{attribute 'pack_mode' := '1'} 
// ------------------------------------------------------------------------- 
//  SRCI Robot Library                                                
// ------------------------------------------------------------------------- 
//                                                                           
//  Object:      vAxesGroupCyclicOptionalDataPlcToRob                                       
//  Author:      Thorsten Brach                                                
//  Date:        2024-06-01
//
//  Description:                                              
//   
//                                                                           
//  Copyright: 
//    (C) 2024 Thorsten Brach. All rights reserved                                                                         
//                                                                           
//  Disclaimer:                                                                           
//    This project is provided without any guarantee and can be used for   
//    private and commercial purposes. Any commercial use is at the user’s 
//    own risk and responsibility.
//
// -------------------------------------------------------------------------
TYPE AxesGroupCyclicOptionalDataPlcToRob :
STRUCT
  /// Transmit cyclic data from PLC to RC for the usage in a subprogram on the RC called via the function “CallSubprogram”
  SubProgramData        :  AxesGroupCyclicOptionalDataSubProgram;
  /// short cartesian position with TCP position (X, Y,Z), rotation (RX, RY, RZ), configuration bytes (Config, TurnNumber), position of first external axis (E1) and corresponding coordinate systems (ToolNo, FrameNo)
  CartesianPosition     :  AxesGroupCyclicOptionalDataCartesianPosition;
  /// the external axis values for an extended cartesian position (E2, E3, E4, E5, E6) 
  /// When selected, Tool and Frame will automatically cyclically be sent from client to server.
  CartesianPositionExt  :  AxesGroupCyclicOptionalDataCartesianPositionExt;
  /// short axes position with joint values (J1, J2, J3,J4, J5, J6) and position of first external axis (E1)
  JointPosition         :  AxesGroupCyclicOptionalDataJointPosition;
  /// the external axis values for an extended joint position (E2, E3, E4, E5, E6)
  JointPositionExt      :  AxesGroupCyclicOptionalDataJointPositionExt;
  /// force with the divided forces in the individual directions (X, Y, Z, RX, RY, RZ)
  CartesianForce        :  AxesGroupCyclicOptionalDataCartesianForce;
  /// current force for the external axis (E1, E2, E3, E4, E5, E6)
  CartesianForceExt     :  AxesGroupCyclicOptionalDataCartesianForceExt;
END_STRUCT
END_TYPE

{attribute 'pack_mode' := '1'} 
// ------------------------------------------------------------------------- 
//  SRCI Robot Library                                                
// ------------------------------------------------------------------------- 
//                                                                           
//  Object:      AxesGroupCyclicOptionalDataRobToPlc                                       
//  Author:      Thorsten Brach                                                
//  Date:        2024-06-01
//
//  Description:                                              
//   
//                                                                           
//  Copyright: 
//    (C) 2024 Thorsten Brach. All rights reserved                                                                         
//                                                                           
//  Disclaimer:                                                                           
//    This project is provided without any guarantee and can be used for   
//    private and commercial purposes. Any commercial use is at the user’s 
//    own risk and responsibility.
//
// -------------------------------------------------------------------------
TYPE AxesGroupCyclicOptionalDataRobToPlc :
STRUCT
  /// Transmit cyclic data from PLC to RC for the usage in a subprogram on the RC called via the function “CallSubprogram”
  SubProgramData        :  AxesGroupCyclicOptionalDataSubProgram;
  /// short cartesian position with TCP position (X, Y,Z), rotation (RX, RY, RZ), configuration bytes (Config, TurnNumber), position of first external axis (E1) and corresponding coordinate systems (ToolNo, FrameNo)
  CartesianPosition     :  AxesGroupCyclicOptionalDataCartesianPosition;
  /// the external axis values for an extended cartesian position (E2, E3, E4, E5, E6) 
  /// When selected, Tool and Frame will automatically cyclically be sent from client to server.
  CartesianPositionExt  :  AxesGroupCyclicOptionalDataCartesianPositionExt;
  /// short axes position with joint values (J1, J2, J3,J4, J5, J6) and position of first external axis (E1)
  JointPosition         :  AxesGroupCyclicOptionalDataJointPosition;
  /// the external axis values for an extended joint position (E2, E3, E4, E5, E6)
  JointPositionExt      :  AxesGroupCyclicOptionalDataJointPositionExt;
  /// force with the divided forces in the individual directions (X, Y, Z, RX, RY, RZ)
  CartesianForce        :  AxesGroupCyclicOptionalDataCartesianForce;
  /// current force for the external axis (E1, E2, E3, E4, E5, E6)
  CartesianForceExt     :  AxesGroupCyclicOptionalDataCartesianForceExt;
  /// ctual axes current of individual axes (J1, J2, J3, J4, J5, J6)
  JointCurrent          :  AxesGroupCyclicOptionalDataJointCurrent;
  /// actual current for the external axis (E1, E2,E3, E4, E5, E6)
  JointCurrentExt       :  AxesGroupCyclicOptionalDataJointCurrentExt;  
END_STRUCT
END_TYPE

{attribute 'pack_mode' := '1'} 
// ------------------------------------------------------------------------- 
//  SRCI Robot Library                                                
// ------------------------------------------------------------------------- 
//                                                                           
//  Object:      AxesGroupCyclic                                       
//  Author:      Thorsten Brach                                                
//  Date:        2024-06-01
//
//  Description:                                              
//   
//                                                                           
//  Copyright: 
//    (C) 2024 Thorsten Brach. All rights reserved                                                                         
//                                                                           
//  Disclaimer:                                                                           
//    This project is provided without any guarantee and can be used for   
//    private and commercial purposes. Any commercial use is at the user’s 
//    own risk and responsibility.
//
// -------------------------------------------------------------------------
TYPE AxesGroupCyclic :
STRUCT
  /// Cyclic data from PLC to Robot 
  PlcToRob : AxesGroupCyclicPlcToRob;
  /// Cyclic data from Robot to PLC
  RobToPlc : AxesGroupCyclicRobToPlc;
END_STRUCT
END_TYPE

{attribute 'pack_mode' := '1'} 
// ------------------------------------------------------------------------- 
//  SRCI Robot Library                                                
// ------------------------------------------------------------------------- 
//                                                                           
//  Object:      AxesGroupCyclicPlcToRob                                       
//  Author:      Thorsten Brach                                                
//  Date:        2024-06-01
//
//  Description:                                              
//   
//                                                                           
//  Copyright: 
//    (C) 2024 Thorsten Brach. All rights reserved                                                                         
//                                                                           
//  Disclaimer:                                                                           
//    This project is provided without any guarantee and can be used for   
//    private and commercial purposes. Any commercial use is at the user’s 
//    own risk and responsibility.
//
// -------------------------------------------------------------------------
TYPE AxesGroupCyclicPlcToRob :
STRUCT
  /// Version of SRCI specification
  /// Bit 0-4 : Minor version = Features        (0..31)
  /// Bit 5-7 : Major version = Breaking change (0..07)
  SRCIVersion            : VersionStruct;
  /// Fast stop trigger 
  FastStop               : BYTE;
  /// Connection alive signal
  LifeSign               : BYTE;
  /// Number of Bytes of the frame to be used for the telegram of the given Axisgroup. Direction client to server
  TelegramLengthPlcToRob : UINT;
  /// Number of Bytes of the frame to be used for the telegram of the given Axisgroup. Direction server to client
  TelegramLengthRobToPlc : UINT;
  /// Control AxesGroupID Telegtam state control
  AxesGroupID            : BYTE;
  /// Telegtam state control
  Control                : ControlHalfByte;
  /// Reserved for later versions
  Reserved               : BYTE;
  /// Configuration of the optional cyclic data. Direction client to server
  TelegramNumberPlcToRob : UINT;
  /// Configuration of the optional cyclic data. Direction server to client
  TelegramNumberRobToPlc : UINT;
  /// Date of the client in the format days since 1990.01.01
  ClientDate             : IEC_DATE;
  /// Time in the clients time zone in the format milliseconds since start of day
  ClientTime             : IEC_TIME;    
END_STRUCT
END_TYPE

{attribute 'pack_mode' := '1'} 
// ------------------------------------------------------------------------- 
//  SRCI Robot Library                                                
// ------------------------------------------------------------------------- 
//                                                                           
//  Object:      AxesGroupCyclicRobToPlc                                       
//  Author:      Thorsten Brach                                                
//  Date:        2024-06-01
//
//  Description:                                              
//   
//                                                                           
//  Copyright: 
//    (C) 2024 Thorsten Brach. All rights reserved                                                                         
//                                                                           
//  Disclaimer:                                                                           
//    This project is provided without any guarantee and can be used for   
//    private and commercial purposes. Any commercial use is at the user’s 
//    own risk and responsibility.
//
// -------------------------------------------------------------------------
TYPE AxesGroupCyclicRobToPlc :
STRUCT
  /// Version of SRCI specification
  /// Bit 0-4 : Minor version = Features        (0..31)
  /// Bit 5-7 : Major version = Breaking change (0..07)
  SRCIVersion   : VersionStruct;
  /// Connection alive signal
  LifeSign      : BYTE;
  /// Reserved byte
  Reserved      : BYTE;
  /// Initialization and Telegram control state
  TelegramState : USINT;
  /// Combination of various RA related states.
  StatusRobotArm: RaStatusWord;
  /// Actual override in percentage encoding 
  Override      : UINT;  
END_STRUCT
END_TYPE

{attribute 'pack_mode' := '1'} 
// ------------------------------------------------------------------------- 
//  SRCI Robot Library                                                
// ------------------------------------------------------------------------- 
//                                                                           
//  Object:      AxesGroupMessageLog                                       
//  Author:      Thorsten Brach                                                
//  Date:        2024-06-01
//
//  Description:                                              
//   
//                                                                           
//  Copyright: 
//    (C) 2024 Thorsten Brach. All rights reserved                                                                         
//                                                                           
//  Disclaimer:                                                                           
//    This project is provided without any guarantee and can be used for   
//    private and commercial purposes. Any commercial use is at the user’s 
//    own risk and responsibility.
//
// -------------------------------------------------------------------------
TYPE AxesGroupMessageLog :
STRUCT
  ///
  SystemLogEntries : UINT := DINT_TO_UINT(RobotLibraryParameter.SYSTEM_LOG_MAX);
  ///
  MessagesEntries  : UINT := DINT_TO_UINT(RobotLibraryParameter.MESSAGE_LOG_MAX);
  ///
  LogLevel         : LogLevel;
  ///
  SystemLog        : ARRAY[0..RobotLibraryParameter.SYSTEM_LOG_MAX] OF STRING(255);
  ///
  Messages         : ARRAY[0..RobotLibraryParameter.MESSAGE_LOG_MAX] OF AlarmMessage;
END_STRUCT
END_TYPE

{attribute 'pack_mode' := '1'} 
// ------------------------------------------------------------------------- 
//  SRCI Robot Library                                                
// ------------------------------------------------------------------------- 
//                                                                           
//  Object:      AxesGroupParameter                                       
//  Author:      Thorsten Brach                                                
//  Date:        2024-06-01
//
//  Description:                                              
//   
//                                                                           
//  Copyright: 
//    (C) 2024 Thorsten Brach. All rights reserved                                                                         
//                                                                           
//  Disclaimer:                                                                           
//    This project is provided without any guarantee and can be used for   
//    private and commercial purposes. Any commercial use is at the user’s 
//    own risk and responsibility.
//
// -------------------------------------------------------------------------
TYPE AxesGroupParameter :
STRUCT
  /// Command parameter
  Cmd            : ARRAY[1..AxesGroupParameterCmdEntries.MAX_ENTRY] OF AxesGroupParameterCmdEntry;
  /// PLC specific data
  Plc            : AxesGroupParameterPlc;
  /// RC data read by the function "ReadRobotData" (see chapter 6.1.2)
  Rob            : AxesGroupParameterRob;
  /// Optional cyclic data configuration
  OptionalCyclic : AxesGroupParameterOptionalCyclic;  
END_STRUCT
END_TYPE

{attribute 'pack_mode' := '1'} 
// ------------------------------------------------------------------------- 
//  SRCI Robot Library                                                
// ------------------------------------------------------------------------- 
//                                                                           
//  Object:      AxesGroupState                                       
//  Author:      Thorsten Brach                                                
//  Date:        2024-06-01
//
//  Description:                                              
//   
//                                                                           
//  Copyright: 
//    (C) 2024 Thorsten Brach. All rights reserved                                                                         
//                                                                           
//  Disclaimer:                                                                           
//    This project is provided without any guarantee and can be used for   
//    private and commercial purposes. Any commercial use is at the user’s 
//    own risk and responsibility.
//
// -------------------------------------------------------------------------
TYPE AxesGroupState :
STRUCT
  ///
  FatalErrorClient  : BOOL;
  ///
  Initialised       : BOOL;
  ///
  Synchronized      : BOOL;
  ///
  Synchronizing     : AxesGroupStateSynchronizing;
  ///
  AliveOk           : BOOL;
  ///
  CMDsEnabled       : BOOL;
  ///
  ConfigExchanged   : BOOL;
  /// 
  RobotIdent        : DT;
  ///
  DataChanged       : AxesGroupStateDataChanged;
  ///
  SyncStatePlc      : AxesGroupStateSyncStatePlc;
  /// 
  SyncStateRc       : AxesGroupStateSyncStateRob;
  ///
  ResetMsg          : AxesGroupStateResetMsg;
  ///
  IncrementFastStop : BOOL;
END_STRUCT
END_TYPE

{attribute 'pack_mode' := '1'} 
// ------------------------------------------------------------------------- 
//  SRCI Robot Library                                                
// ------------------------------------------------------------------------- 
//                                                                           
//  Object:      TelegramPlcToRob                                       
//  Author:      Thorsten Brach                                                
//  Date:        2024-06-01
//
//  Description:                                              
//   
//                                                                           
//  Copyright: 
//    (C) 2024 Thorsten Brach. All rights reserved                                                                         
//                                                                           
//  Disclaimer:                                                                           
//    This project is provided without any guarantee and can be used for   
//    private and commercial purposes. Any commercial use is at the user’s 
//    own risk and responsibility.
//
// -------------------------------------------------------------------------
TYPE TelegramPlcToRob :
STRUCT
  /// Header
  Header              : TelegramPlcToRobHeader;
  /// Cyclic data 
  //Cyclic               : TelegramPlcToRobCyclic;
  /// Cyclic optional data
  CyclicOptional       : TelegramPlcToRobCyclicOptionalData;
  /// Sequence Data
  Sequence             : ARRAY[0..1] OF TelegramPlcToRobSequence;
  /// Footer
  Footer               : TelegramFooter;
END_STRUCT
END_TYPE

{attribute 'pack_mode' := '1'} 
// ------------------------------------------------------------------------- 
//  SRCI Robot Library                                                
// ------------------------------------------------------------------------- 
//                                                                           
//  Object:      TelegramRobToPlc                                       
//  Author:      Thorsten Brach                                                
//  Date:        2024-06-01
//
//  Description:                                              
//   
//                                                                           
//  Copyright: 
//    (C) 2024 Thorsten Brach. All rights reserved                                                                         
//                                                                           
//  Disclaimer:                                                                           
//    This project is provided without any guarantee and can be used for   
//    private and commercial purposes. Any commercial use is at the user’s 
//    own risk and responsibility.
//
// -------------------------------------------------------------------------
TYPE TelegramRobToPlc :
STRUCT
  /// Telegram Header
  Header               : TelegramRobToPlcHeader;
  /// Cyclic optional data
  CyclicOptional       : TelegramRobToPlcCyclicOptionalData;
  /// Sequence Data
  Sequence             : ARRAY[0..1] OF TelegramPlcToRobSequence;
  /// Footer
  Footer               : TelegramFooter;
END_STRUCT
END_TYPE

{attribute 'pack_mode' := '1'} 
// ------------------------------------------------------------------------- 
//  SRCI Robot Library                                                
// ------------------------------------------------------------------------- 
//                                                                           
//  Object:      AxesGroupCyclicOptionalDataCartesianForce                                       
//  Author:      Thorsten Brach                                                
//  Date:        2024-06-01
//
//  Description:                                              
//   
//                                                                           
//  Copyright: 
//    (C) 2024 Thorsten Brach. All rights reserved                                                                         
//                                                                           
//  Disclaimer:                                                                           
//    This project is provided without any guarantee and can be used for   
//    private and commercial purposes. Any commercial use is at the user’s 
//    own risk and responsibility.
//
// -------------------------------------------------------------------------
TYPE AxesGroupCyclicOptionalDataCartesianForce EXTENDS RobotCartesianForceShort:
STRUCT
  /// indicates that this optional parameter will be used
  Active           : BOOL;
END_STRUCT
END_TYPE

{attribute 'pack_mode' := '1'} 
// ------------------------------------------------------------------------- 
//  SRCI Robot Library                                                
// ------------------------------------------------------------------------- 
//                                                                           
//  Object:      AxesGroupCyclicOptionalDataCartesianForceExt                                       
//  Author:      Thorsten Brach                                                
//  Date:        2024-06-01
//
//  Description:                                              
//   
//                                                                           
//  Copyright: 
//    (C) 2024 Thorsten Brach. All rights reserved                                                                         
//                                                                           
//  Disclaimer:                                                                           
//    This project is provided without any guarantee and can be used for   
//    private and commercial purposes. Any commercial use is at the user’s 
//    own risk and responsibility.
//
// -------------------------------------------------------------------------
TYPE AxesGroupCyclicOptionalDataCartesianForceExt EXTENDS RobotCartesianForceExt:
STRUCT
  /// indicates that this optional parameter will be used
  Active           : BOOL;
END_STRUCT
END_TYPE

{attribute 'pack_mode' := '1'} 
// ------------------------------------------------------------------------- 
//  SRCI Robot Library                                                
// ------------------------------------------------------------------------- 
//                                                                           
//  Object:      AxesGroupCyclicOptionalDataCartesianPosition                                       
//  Author:      Thorsten Brach                                                
//  Date:        2024-06-01
//
//  Description:                                              
//   
//                                                                           
//  Copyright: 
//    (C) 2024 Thorsten Brach. All rights reserved                                                                         
//                                                                           
//  Disclaimer:                                                                           
//    This project is provided without any guarantee and can be used for   
//    private and commercial purposes. Any commercial use is at the user’s 
//    own risk and responsibility.
//
// -------------------------------------------------------------------------
TYPE AxesGroupCyclicOptionalDataCartesianPosition EXTENDS  RobotCartesianPositionShort :
STRUCT
  /// indicates that this optional parameter will be used
  Active           : BOOL;
  /// corresponding coordinate systems
  CoordinateSystem : RobotCoordinateSystemParameters; 
END_STRUCT
END_TYPE

{attribute 'pack_mode' := '1'} 
// ------------------------------------------------------------------------- 
//  SRCI Robot Library                                                
// ------------------------------------------------------------------------- 
//                                                                           
//  Object:      AxesGroupCyclicOptionalDataCartesianPositionExt                                       
//  Author:      Thorsten Brach                                                
//  Date:        2024-06-01
//
//  Description:                                              
//   
//                                                                           
//  Copyright: 
//    (C) 2024 Thorsten Brach. All rights reserved                                                                         
//                                                                           
//  Disclaimer:                                                                           
//    This project is provided without any guarantee and can be used for   
//    private and commercial purposes. Any commercial use is at the user’s 
//    own risk and responsibility.
//
// -------------------------------------------------------------------------
TYPE AxesGroupCyclicOptionalDataCartesianPositionExt EXTENDS RobotCartesianPositionExt :
STRUCT
  /// indicates that this optional parameter will be used
  Active : BOOL;
END_STRUCT
END_TYPE

{attribute 'pack_mode' := '1'} 
// ------------------------------------------------------------------------- 
//  SRCI Robot Library                                                
// ------------------------------------------------------------------------- 
//                                                                           
//  Object:      AxesGroupCyclicOptionalDataJointCurrent                                       
//  Author:      Thorsten Brach                                                
//  Date:        2024-06-01
//
//  Description:                                              
//   
//                                                                           
//  Copyright: 
//    (C) 2024 Thorsten Brach. All rights reserved                                                                         
//                                                                           
//  Disclaimer:                                                                           
//    This project is provided without any guarantee and can be used for   
//    private and commercial purposes. Any commercial use is at the user’s 
//    own risk and responsibility.
//
// -------------------------------------------------------------------------
TYPE AxesGroupCyclicOptionalDataJointCurrent EXTENDS RobotJointCurrentShort :
STRUCT
    /// indicates that this optional parameter will be used
  Active : BOOL;
END_STRUCT
END_TYPE

{attribute 'pack_mode' := '1'} 
// ------------------------------------------------------------------------- 
//  SRCI Robot Library                                                
// ------------------------------------------------------------------------- 
//                                                                           
//  Object:      AxesGroupCyclicOptionalDataJointCurrentExt                                       
//  Author:      Thorsten Brach                                                
//  Date:        2024-06-01
//
//  Description:                                              
//   
//                                                                           
//  Copyright: 
//    (C) 2024 Thorsten Brach. All rights reserved                                                                         
//                                                                           
//  Disclaimer:                                                                           
//    This project is provided without any guarantee and can be used for   
//    private and commercial purposes. Any commercial use is at the user’s 
//    own risk and responsibility.
//
// -------------------------------------------------------------------------
TYPE AxesGroupCyclicOptionalDataJointCurrentExt EXTENDS RobotJointCurrentExt :
STRUCT
    /// indicates that this optional parameter will be used
  Active : BOOL;
END_STRUCT
END_TYPE

{attribute 'pack_mode' := '1'} 
// ------------------------------------------------------------------------- 
//  SRCI Robot Library                                                
// ------------------------------------------------------------------------- 
//                                                                           
//  Object:      AxesGroupCyclicOptionalDataJointPosition                                       
//  Author:      Thorsten Brach                                                
//  Date:        2024-06-01
//
//  Description:                                              
//   
//                                                                           
//  Copyright: 
//    (C) 2024 Thorsten Brach. All rights reserved                                                                         
//                                                                           
//  Disclaimer:                                                                           
//    This project is provided without any guarantee and can be used for   
//    private and commercial purposes. Any commercial use is at the user’s 
//    own risk and responsibility.
//
// -------------------------------------------------------------------------
TYPE AxesGroupCyclicOptionalDataJointPosition EXTENDS RobotJointPositionShort :
STRUCT
    /// indicates that this optional parameter will be used
  Active : BOOL;
END_STRUCT
END_TYPE

{attribute 'pack_mode' := '1'} 
// ------------------------------------------------------------------------- 
//  SRCI Robot Library                                                
// ------------------------------------------------------------------------- 
//                                                                           
//  Object:      AxesGroupCyclicOptionalDataJointPositionExt                                       
//  Author:      Thorsten Brach                                                
//  Date:        2024-06-01
//
//  Description:                                              
//   
//                                                                           
//  Copyright: 
//    (C) 2024 Thorsten Brach. All rights reserved                                                                         
//                                                                           
//  Disclaimer:                                                                           
//    This project is provided without any guarantee and can be used for   
//    private and commercial purposes. Any commercial use is at the user’s 
//    own risk and responsibility.
//
// -------------------------------------------------------------------------
TYPE AxesGroupCyclicOptionalDataJointPositionExt EXTENDS RobotJointPositionExt :
STRUCT
    /// indicates that this optional parameter will be used
  Active : BOOL;
END_STRUCT
END_TYPE

{attribute 'pack_mode' := '1'} 
// ------------------------------------------------------------------------- 
//  SRCI Robot Library                                                
// ------------------------------------------------------------------------- 
//                                                                           
//  Object:      AxesGroupCyclicOptionalDataSubProgram                                       
//  Author:      Thorsten Brach                                                
//  Date:        2024-06-01
//
//  Description:                                              
//   
//                                                                           
//  Copyright: 
//    (C) 2024 Thorsten Brach. All rights reserved                                                                         
//                                                                           
//  Disclaimer:                                                                           
//    This project is provided without any guarantee and can be used for   
//    private and commercial purposes. Any commercial use is at the user’s 
//    own risk and responsibility.
//
// -------------------------------------------------------------------------
TYPE AxesGroupCyclicOptionalDataSubProgram EXTENDS RobotSubProgramData :
STRUCT
  /// indicates that this optional parameter will be used
  Active : BOOL;
END_STRUCT
END_TYPE

{attribute 'pack_mode' := '1'} 
// ------------------------------------------------------------------------- 
//  SRCI Robot Library                                                
// ------------------------------------------------------------------------- 
//                                                                           
//  Object:      AxesGroupParameterCmdEntry                                       
//  Author:      Thorsten Brach                                                
//  Date:        2024-06-01
//
//  Description:                                              
//   
//                                                                           
//  Copyright: 
//    (C) 2024 Thorsten Brach. All rights reserved                                                                         
//                                                                           
//  Disclaimer:                                                                           
//    This project is provided without any guarantee and can be used for   
//    private and commercial purposes. Any commercial use is at the user’s 
//    own risk and responsibility.
//
// -------------------------------------------------------------------------
TYPE AxesGroupParameterCmdEntry :
STRUCT
  /// User defined command name
  Name                 : STRING(20);
  ///
  CmdType              : CmdType; 
  ///
  Prio                 : PriorityLevel;
  ///
  HighPrio             : USINT;
  ///
  ExecMode             : ExecutionMode;
  ///
  SequenceFlag         : SequenceFlag;
  /// ID of Action that will be executed when this command is active
  /// • >0: Start Action - Start executing the Action function with the identical ListenerID.
  /// • <0: Stop Action  -  Stop executing the Action function with the identical ListenerID.
  /// • 0: No trigger (default)-  If no EmitterID is defined, the function will not trigger any Action during its execution
  /// For more information see section Triggers of this chapter or chapter 5.5.12.4.
  EmitterID            : ARRAY [0..3] OF SINT;
  /// ID of associated trigger function:
  /// • 0: No Trigger (default): No trigger related behavior
  /// • >0: Trigger:  Start executing, when the trigger function with the identical EmitterID is triggered.
  /// Always positive.
  /// For more information, see chapter 5.5.12 Triggers
  ListenerID           : SINT;
  ///
  ExecutionModeAllowed : ProcessingModeAllowed;
  ///
  LogParameter         : LogParameter;
  ///
  FunctionMode         : USINT; // ToDo ?
  ///
  CheckEmitterID       : SINT;
  ///
  CheckListenerID      : SINT;
END_STRUCT
END_TYPE

{attribute 'pack_mode' := '1'} 
// ------------------------------------------------------------------------- 
//  SRCI Robot Library                                                
// ------------------------------------------------------------------------- 
//                                                                           
//  Object:      AxesGroupParameterOptionalCyclic                                       
//  Author:      Thorsten Brach                                                
//  Date:        2024-06-01
//
//  Description:                                              
//   
//                                                                           
//  Copyright: 
//    (C) 2024 Thorsten Brach. All rights reserved                                                                         
//                                                                           
//  Disclaimer:                                                                           
//    This project is provided without any guarantee and can be used for   
//    private and commercial purposes. Any commercial use is at the user’s 
//    own risk and responsibility.
//
// -------------------------------------------------------------------------
TYPE AxesGroupParameterOptionalCyclic :
STRUCT
  /// Configuration of optional cyclic data send to the Robot
  PlcToRob : AxesGroupParameterOptionalCyclicPlcToRob;
  /// Configuration of optional cyclic data received from the Robot
  RobToPlc : AxesGroupParameterOptionalCyclicRobToPlc;
END_STRUCT
END_TYPE

{attribute 'pack_mode' := '1'} 
// ------------------------------------------------------------------------- 
//  SRCI Robot Library                                                
// ------------------------------------------------------------------------- 
//                                                                           
//  Object:      AxesGroupParameterOptionalCyclicPlcToRob                                       
//  Author:      Thorsten Brach                                                
//  Date:        2024-06-01
//
//  Description:                                              
//   
//                                                                           
//  Copyright: 
//    (C) 2024 Thorsten Brach. All rights reserved                                                                         
//                                                                           
//  Disclaimer:                                                                           
//    This project is provided without any guarantee and can be used for   
//    private and commercial purposes. Any commercial use is at the user’s 
//    own risk and responsibility.
//
// -------------------------------------------------------------------------
TYPE AxesGroupParameterOptionalCyclicPlcToRob :
STRUCT
  /// Bit 00: 
  /// Transmit cyclic data from PLC to RC for the usage in a subprogram on the RC called via the function “CallSubprogram”
  UseCallSubprogram       : BOOL;
  /// Bit 01: 
  /// Send a short cartesian position with TCP position (X, Y,Z), rotation (RX, RY, RZ), 
  /// configuration bytes (Config, TurnNumber), position of first external axis (E1) and corresponding coordinate systems (ToolNo, FrameNo)
  UseCartesianPos         : BOOL;
  /// Bit 02: 
  /// Send a short axes position with joint values (J1, J2, J3, J4, J5, J6) and position of first external axis (E1)
  UseJointPos             : BOOL;
  /// Bit 03: 
  /// Send the force with the divided forces in the individual directions (X, Y, Z, RX, RY, RZ)
  UseForce                : BOOL;
  /// Bit 04:
  Bit04                   : BOOL;
  /// Bit 05:
  Bit05                   : BOOL;
  /// Bit 06:
  Bit06                   : BOOL;
  /// Bit 07:
  Bit07                   : BOOL;  
  /// Bit 08: 
  /// Set to 1 to define two Sequences in one Telegram. 
  /// If activated, 2 sequences also has to be activated in the ServerClient direction
  UseTwoSequences         : BOOL;
  /// Bit 09: 
  /// Send the external axis values for an extended cartesian position (E2, E3, E4, E5, E6)
  UseCartesianPositionExt : BOOL;
  /// Bit 10: 
  /// Send the external axis values for an extended joint position (E2, E3, E4, E5, E6)
  UseJointPositionExt     : BOOL;
  /// Bit 11:
  Bit11                   : BOOL;
  /// Bit 12:
  Bit12                   : BOOL;
  /// Bit 13:
  Bit13                   : BOOL;
  /// Bit 14:
  Bit14                   : BOOL;
  /// Bit 15:
  Bit15                   : BOOL;  
END_STRUCT
END_TYPE

{attribute 'pack_mode' := '1'} 
// ------------------------------------------------------------------------- 
//  SRCI Robot Library                                                
// ------------------------------------------------------------------------- 
//                                                                           
//  Object:      AxesGroupParameterOptionalCyclicRobToPlc                                       
//  Author:      Thorsten Brach                                                
//  Date:        2024-06-01
//
//  Description:                                              
//   
//                                                                           
//  Copyright: 
//    (C) 2024 Thorsten Brach. All rights reserved                                                                         
//                                                                           
//  Disclaimer:                                                                           
//    This project is provided without any guarantee and can be used for   
//    private and commercial purposes. Any commercial use is at the user’s 
//    own risk and responsibility.
//
// -------------------------------------------------------------------------
TYPE AxesGroupParameterOptionalCyclicRobToPlc :
STRUCT
  /// Bit 00: 
  /// Transmit cyclic data from PLC to RC for the usage in a subprogram on the RC called via the function “CallSubprogram”
  UseCallSubprogram       : BOOL;
  /// Bit 01: 
  /// Send a short cartesian position with TCP position (X, Y,Z), rotation (RX, RY, RZ), 
  /// configuration bytes (Config, TurnNumber), position of first external axis (E1) and corresponding coordinate systems (ToolNo, FrameNo)
  UseCartesianPos         : BOOL;
  /// Bit 02: 
  /// Send a short axes position with joint values (J1, J2, J3, J4, J5, J6) and position of first external axis (E1)
  UseJointPos             : BOOL;
  /// Bit 03: 
  /// Send the force with the divided forces in the individual directions (X, Y, Z, RX, RY, RZ)
  UseForce                : BOOL;
  /// Bit 04:
  /// Transmit actual axes current of individual axes (J1, J2, J3, J4, J5, J6)
  UseCurrent              : BOOL;
  /// Bit 05:
  Bit05                   : BOOL;
  /// Bit 06:
  Bit06                   : BOOL;
  /// Bit 07:
  Bit07                   : BOOL;  
  /// Bit 08: 
  /// Set to 1 to define two Sequences in one Telegram. 
  /// If activated, 2 sequences also has to be activated in the ServerClient direction
  UseTwoSequences         : BOOL;
  /// Bit 09: 
  /// Send the external axis values for an extended cartesian position (E2, E3, E4, E5, E6)
  UseCartesianPositionExt : BOOL;
  /// Bit 10: 
  /// Send the external axis values for an extended joint position (E2, E3, E4, E5, E6)
  UseJointPositionExt     : BOOL;
  /// Bit 11:
  /// Transmit the current force for the external axis (E1, E2, E3, E4, E5, E6)
  UseForceExt             : BOOL;
  /// Bit 12:
  /// Transmit the actual current for the external axis (E1, E2, E3, E4, E5, E6)
  UseCurrentEct           : BOOL;
  /// Bit 13:
  Bit13                   : BOOL;
  /// Bit 14:
  Bit14                   : BOOL;
  /// Bit 15:
  Bit15                   : BOOL;  
END_STRUCT
END_TYPE

{attribute 'pack_mode' := '1'} 
// ------------------------------------------------------------------------- 
//  SRCI Robot Library                                                
// ------------------------------------------------------------------------- 
//                                                                           
//  Object:      AxesGroupParameterPlc                                       
//  Author:      Thorsten Brach                                                
//  Date:        2024-06-01
//
//  Description:                                              
//   
//                                                                           
//  Copyright: 
//    (C) 2024 Thorsten Brach. All rights reserved                                                                         
//                                                                           
//  Disclaimer:                                                                           
//    This project is provided without any guarantee and can be used for   
//    private and commercial purposes. Any commercial use is at the user’s 
//    own risk and responsibility.
//
// -------------------------------------------------------------------------
TYPE AxesGroupParameterPlc :
STRUCT
  /// Manufactured ID
  ManufacturedID       : UINT;
  /// Order ID
  OrderID              : STRING(20);
  /// Serial Number
  SerialNumber         : STRING(16);
  /// Firmware Version
  FirmwareVersion      : STRING(8);
  /// Client Interface Version
  InterfaceVersion     : STRING(8);
  /// Synchronization Modes
  SynchronizationModes : SynchronizationModes;  
END_STRUCT
END_TYPE

{attribute 'pack_mode' := '1'} 
// ------------------------------------------------------------------------- 
//  SRCI Robot Library                                                
// ------------------------------------------------------------------------- 
//                                                                           
//  Object:      AxesGroupParameterRob                                       
//  Author:      Thorsten Brach                                                
//  Date:        2024-06-01
//
//  Description:                                              
//   
//                                                                           
//  Copyright: 
//    (C) 2024 Thorsten Brach. All rights reserved                                                                         
//                                                                           
//  Disclaimer:                                                                           
//    This project is provided without any guarantee and can be used for   
//    private and commercial purposes. Any commercial use is at the user’s 
//    own risk and responsibility.
//
// -------------------------------------------------------------------------
TYPE AxesGroupParameterRob :
STRUCT  
  /// User defined robot name
  RobotName       : STRING(20);
  ///  Size of (A)ctive (C)ommand (R)egister
  AcrSize         : UINT;
  /// Ammount of RC managed tools
  ToolCount       : USINT;
  /// Ammount of RC managed frames 
  FrameCount      : USINT;
  /// Ammount of RC managed load data 
  LoadCount       : USINT;
  /// Ammount of RC managed work areas 
  WorkAreaCount   : USINT;
  /// Ammount of working hours of the robot control
  WorkingHoursRc  : UDINT;
  /// Ammount of working hours of the robot arm
  WorkingHoursRa  : UDINT;
END_STRUCT
END_TYPE

{attribute 'pack_mode' := '1'} 
// ------------------------------------------------------------------------- 
//  SRCI Robot Library                                                
// ------------------------------------------------------------------------- 
//                                                                           
//  Object:      AxesGroupStateDataChanged                                       
//  Author:      Thorsten Brach                                                
//  Date:        2024-06-01
//
//  Description:                                              
//   
//                                                                           
//  Copyright: 
//    (C) 2024 Thorsten Brach. All rights reserved                                                                         
//                                                                           
//  Disclaimer:                                                                           
//    This project is provided without any guarantee and can be used for   
//    private and commercial purposes. Any commercial use is at the user’s 
//    own risk and responsibility.
//
// -------------------------------------------------------------------------
TYPE AxesGroupStateDataChanged :
STRUCT
  /// indicates that tool data has changed
  Tool             : ARRAY[0..255] OF BOOL;
  /// indicates that frame data has changed
  Frame            : ARRAY[0..255] OF BOOL;
  /// indicates that load data has changed
  Load             : ARRAY[0..255] OF BOOL;
  /// indicates that work area has changed
  WorkArea         : ARRAY[0..255] OF BOOL;
  /// indicates that default dynamic has changed
  DefaultDynamic   : BOOL;
  /// indicates that reference dynamic has changed
  ReferenceDynamic : BOOL;
  /// indicates that software limits has changed
  SwLimits         : BOOL;
END_STRUCT
END_TYPE

{attribute 'pack_mode' := '1'} 
// ------------------------------------------------------------------------- 
//  SRCI Robot Library                                                
// ------------------------------------------------------------------------- 
//                                                                           
//  Object:      AxesGroupStateResetMsg                                       
//  Author:      Thorsten Brach                                                
//  Date:        2024-06-01
//
//  Description:                                              
//   
//                                                                           
//  Copyright: 
//    (C) 2024 Thorsten Brach. All rights reserved                                                                         
//                                                                           
//  Disclaimer:                                                                           
//    This project is provided without any guarantee and can be used for   
//    private and commercial purposes. Any commercial use is at the user’s 
//    own risk and responsibility.
//
// -------------------------------------------------------------------------
TYPE AxesGroupStateResetMsg :
STRUCT
  ///
  Reset     : BOOL;
  ///
  ResetTime : DT;
END_STRUCT
END_TYPE

{attribute 'pack_mode' := '1'} 
// ------------------------------------------------------------------------- 
//  SRCI Robot Library                                                
// ------------------------------------------------------------------------- 
//                                                                           
//  Object:      AxesGroupStateSynchronizing                                       
//  Author:      Thorsten Brach                                                
//  Date:        2024-06-01
//
//  Description:                                              
//   
//                                                                           
//  Copyright: 
//    (C) 2024 Thorsten Brach. All rights reserved                                                                         
//                                                                           
//  Disclaimer:                                                                           
//    This project is provided without any guarantee and can be used for   
//    private and commercial purposes. Any commercial use is at the user’s 
//    own risk and responsibility.
//
// -------------------------------------------------------------------------
TYPE AxesGroupStateSynchronizing :
STRUCT
  /// indicates that the tooldata are synchronized
  Tool           : BOOL;
  /// indicates that the framedata are synchronized
  Frame          : BOOL;
  /// indicates that the loaddata are synchronized
  Load           : BOOL;
  /// indicates that the work areas are synchronized
  WorkAreas      : BOOL;
  /// indicates that the reference-dynamics are synchronized
  RefDynamic     : BOOL;
  /// indicates that the default-dynamics are synchronized
  DefaultDynamic : BOOL;
  /// indicates that the software limits are synchronized
  SwLimits       : BOOL;
END_STRUCT
END_TYPE

{attribute 'pack_mode' := '1'} 
// ------------------------------------------------------------------------- 
//  SRCI Robot Library                                                
// ------------------------------------------------------------------------- 
//                                                                           
//  Object:      AxesGroupStateSyncState                                       
//  Author:      Thorsten Brach                                                
//  Date:        2024-06-01
//
//  Description:                                              
//   
//                                                                           
//  Copyright: 
//    (C) 2024 Thorsten Brach. All rights reserved                                                                         
//                                                                           
//  Disclaimer:                                                                           
//    This project is provided without any guarantee and can be used for   
//    private and commercial purposes. Any commercial use is at the user’s 
//    own risk and responsibility.
//
// -------------------------------------------------------------------------
TYPE AxesGroupStateSyncState :
STRUCT
  /// Bit 00: Tool
  Tool             : BOOL;
  /// Bit 01: Frame
  Frame            : BOOL;
  /// Bit 02: Load
  Load             : BOOL;
  /// Bit 03: WorkArea
  WorkArea         : BOOL;
  /// Bit 04: SwLimits
  SwLimits         : BOOL;
  /// Bit 05: DefaultDynamic
  DefaultDynamic   : BOOL;
  /// Bit 06: ReferenceDynamic
  ReferenceDynamic : BOOL;
  /// Bit 07:
  Bit07            : BOOL;
  /// Bit 08:
  Bit08            : BOOL;
  /// Bit 09:
  Bit09            : BOOL;
  /// Bit 10:
  Bit10            : BOOL;
  /// Bit 11:
  Bit11            : BOOL;
  /// Bit 12:
  Bit12            : BOOL;
  /// Bit 13:
  Bit13            : BOOL;
  /// Bit 14:
  Bit14            : BOOL;
  /// Bit 15:
  Bit15            : BOOL;  
END_STRUCT
END_TYPE

{attribute 'pack_mode' := '1'} 
// ------------------------------------------------------------------------- 
//  SRCI Robot Library                                                
// ------------------------------------------------------------------------- 
//                                                                           
//  Object:      AxesGroupStateSyncStateNo                                       
//  Author:      Thorsten Brach                                                
//  Date:        2024-06-01
//
//  Description:                                              
//   
//                                                                           
//  Copyright: 
//    (C) 2024 Thorsten Brach. All rights reserved                                                                         
//                                                                           
//  Disclaimer:                                                                           
//    This project is provided without any guarantee and can be used for   
//    private and commercial purposes. Any commercial use is at the user’s 
//    own risk and responsibility.
//
// -------------------------------------------------------------------------
TYPE AxesGroupStateSyncStateNo :
STRUCT
  /// Ammount of unsynchronized tool data
  Tool     : USINT;
  /// Ammount of unsynchronized frame data
  Frame    : USINT;
  /// Ammount of unsynchronized load data
  Load     : USINT;
  /// Ammount of unsynchronized word areas
  WorkArea : USINT;    
END_STRUCT
END_TYPE

{attribute 'pack_mode' := '1'} 
// ------------------------------------------------------------------------- 
//  SRCI Robot Library                                                
// ------------------------------------------------------------------------- 
//                                                                           
//  Object:      AxesGroupStateSyncStatePlc                                       
//  Author:      Thorsten Brach                                                
//  Date:        2024-06-01
//
//  Description:                                              
//   
//                                                                           
//  Copyright: 
//    (C) 2024 Thorsten Brach. All rights reserved                                                                         
//                                                                           
//  Disclaimer:                                                                           
//    This project is provided without any guarantee and can be used for   
//    private and commercial purposes. Any commercial use is at the user’s 
//    own risk and responsibility.
//
// -------------------------------------------------------------------------
TYPE AxesGroupStateSyncStatePlc :
STRUCT
  ///
  InSync   : AxesGroupStateSyncState;
END_STRUCT
END_TYPE

{attribute 'pack_mode' := '1'} 
// ------------------------------------------------------------------------- 
//  SRCI Robot Library                                                
// ------------------------------------------------------------------------- 
//                                                                           
//  Object:      AxesGroupStateSyncStateRob                                       
//  Author:      Thorsten Brach                                                
//  Date:        2024-06-01
//
//  Description:                                              
//   
//                                                                           
//  Copyright: 
//    (C) 2024 Thorsten Brach. All rights reserved                                                                         
//                                                                           
//  Disclaimer:                                                                           
//    This project is provided without any guarantee and can be used for   
//    private and commercial purposes. Any commercial use is at the user’s 
//    own risk and responsibility.
//
// -------------------------------------------------------------------------
TYPE AxesGroupStateSyncStateRob :
STRUCT
  ///
  InSync   : AxesGroupStateSyncState;
  ///
  UnSyncNo : AxesGroupStateSyncStateNo;
END_STRUCT
END_TYPE

{attribute 'pack_mode' := '1'} 
// ------------------------------------------------------------------------- 
//  SRCI Robot Library                                                
// ------------------------------------------------------------------------- 
//                                                                           
//  Object:      TelegramPlcToRobMessage                                       
//  Author:      Thorsten Brach                                                
//  Date:        2024-06-01
//
//  Description:                                              
//   
//                                                                           
//  Copyright: 
//    (C) 2024 Thorsten Brach. All rights reserved                                                                         
//                                                                           
//  Disclaimer:                                                                           
//    This project is provided without any guarantee and can be used for   
//    private and commercial purposes. Any commercial use is at the user’s 
//    own risk and responsibility.
//
// -------------------------------------------------------------------------
TYPE TelegramPlcToRobCommand :
STRUCT
  /// Header
  Header  : TelegramPlcToRobCommandHeader;
  /// Payload
  Payload : ARRAY[1..255] OF BYTE; // ToDo
END_STRUCT
END_TYPE

{attribute 'pack_mode' := '1'} 
// ------------------------------------------------------------------------- 
//  SRCI Robot Library                                                
// ------------------------------------------------------------------------- 
//                                                                           
//  Object:      TelegramPlcToRobMessageHeader                                       
//  Author:      Thorsten Brach                                                
//  Date:        2024-06-01
//
//  Description:                                              
//   
//                                                                           
//  Copyright: 
//    (C) 2024 Thorsten Brach. All rights reserved                                                                         
//                                                                           
//  Disclaimer:                                                                           
//    This project is provided without any guarantee and can be used for   
//    private and commercial purposes. Any commercial use is at the user’s 
//    own risk and responsibility.
//
// -------------------------------------------------------------------------
TYPE TelegramPlcToRobCommandHeader :
STRUCT
  /// Command type
  CmdType           : CmdType;
  /// CMD priority level
  Prio              : PriorityLevel;
  /// Execution Mode
  ExecMode          : ExecutionMode;
  /// Parameter Sequence
  ParSequence       : BYTE;
END_STRUCT
END_TYPE

{attribute 'pack_mode' := '1'} 
// ------------------------------------------------------------------------- 
//  SRCI Robot Library                                                
// ------------------------------------------------------------------------- 
//                                                                           
//  Object:      TelegramPlcToRobCyclicOptionalData                                       
//  Author:      Thorsten Brach                                                
//  Date:        2024-06-01
//
//  Description:                                              
//   
//                                                                           
//  Copyright: 
//    (C) 2024 Thorsten Brach. All rights reserved                                                                         
//                                                                           
//  Disclaimer:                                                                           
//    This project is provided without any guarantee and can be used for   
//    private and commercial purposes. Any commercial use is at the user’s 
//    own risk and responsibility.
//
// -------------------------------------------------------------------------
TYPE TelegramPlcToRobCyclicOptionalData :
STRUCT
  /// Transmit cyclic data from PLC to RC for the usage in a subprogram on the RC called via the function “CallSubprogram”
  SubProgramData        :  TelegramPlcToRobCyclicOptionalSubProgramData;
  /// short cartesian position with TCP position (X, Y,Z), rotation (RX, RY, RZ), configuration bytes (Config, TurnNumber), position of first external axis (E1) and corresponding coordinate systems (ToolNo, FrameNo)
  CartesianPos          :  TelegramPlcToRobCyclicOptionalCartesianPosition;
  /// the external axis values for an extended cartesian position (E2, E3, E4, E5, E6) 
  /// When selected, Tool and Frame will automatically cyclically be sent from client to server.
  CartesianPosExt       :  TelegramPlcToRobCyclicOptionalCartesianPositionExt;
  /// short axes position with joint values (J1, J2, J3,J4, J5, J6) and position of first external axis (E1)
  JointPosition         :  TelegramPlcToRobCyclicOptionalJointPosition;
  /// the external axis values for an extended joint position (E2, E3, E4, E5, E6)
  JointPositionExt      :  TelegramPlcToRobCyclicOptionalJointPositionExt;
  /// force with the divided forces in the individual directions (X, Y, Z, RX, RY, RZ)
  Force                 :  TelegramPlcToRobCyclicOptionalForce;
  /// current force for the external axis (E1, E2, E3, E4, E5, E6)
  ForceExt              :  TelegramPlcToRobCyclicOptionalForceExt;
  /// ctual axes current of individual axes (J1, J2, J3, J4, J5, J6)
  Current               :  TelegramPlcToRobCyclicOptionalCurrent;
  /// actual current for the external axis (E1, E2,E3, E4, E5, E6)
  CurrentExt            :  TelegramPlcToRobCyclicOptionalCurrentExt;
END_STRUCT
END_TYPE

{attribute 'pack_mode' := '1'} 
// ------------------------------------------------------------------------- 
//  SRCI Robot Library                                                
// ------------------------------------------------------------------------- 
//                                                                           
//  Object:      TelegramPlcToRobFooter                                       
//  Author:      Thorsten Brach                                                
//  Date:        2024-06-01
//
//  Description:                                              
//   
//                                                                           
//  Copyright: 
//    (C) 2024 Thorsten Brach. All rights reserved                                                                         
//                                                                           
//  Disclaimer:                                                                           
//    This project is provided without any guarantee and can be used for   
//    private and commercial purposes. Any commercial use is at the user’s 
//    own risk and responsibility.
//
// -------------------------------------------------------------------------
TYPE TelegramPlcToRobFooter :
STRUCT
  /// Bit 00: Connection alive signal
  LifeSign : BOOL;
  /// Bit 01 
  Bit01    : BOOL;
  /// Bit 02 
  Bit02    : BOOL;
  /// Bit 03 
  Bit03    : BOOL;
  /// Bit 04 
  Bit04    : BOOL;
  /// Bit 05 
  Bit05    : BOOL;
  /// Bit 06 
  Bit06    : BOOL;
  /// Bit 07 
  Bit07    : BOOL;  
END_STRUCT
END_TYPE

{attribute 'pack_mode' := '1'} 
// ------------------------------------------------------------------------- 
//  SRCI Robot Library                                                
// ------------------------------------------------------------------------- 
//                                                                           
//  Object:      TelegramPlcToRobFragment                                       
//  Author:      Thorsten Brach                                                
//  Date:        2024-06-01
//
//  Description:                                              
//   
//                                                                           
//  Copyright: 
//    (C) 2024 Thorsten Brach. All rights reserved                                                                         
//                                                                           
//  Disclaimer:                                                                           
//    This project is provided without any guarantee and can be used for   
//    private and commercial purposes. Any commercial use is at the user’s 
//    own risk and responsibility.
//
// -------------------------------------------------------------------------
TYPE TelegramPlcToRobFragment :
STRUCT
  /// Header
  Header  : TelegramPlcToRobFragmentHeader;
  /// Command
  Command : TelegramPlcToRobCommand;
END_STRUCT
END_TYPE

{attribute 'pack_mode' := '1'} 
// ------------------------------------------------------------------------- 
//  SRCI Robot Library                                                
// ------------------------------------------------------------------------- 
//                                                                           
//  Object:      TelegramPlcToRobFragmentHeader                                       
//  Author:      Thorsten Brach                                                
//  Date:        2024-06-01
//
//  Description:                                              
//   
//                                                                           
//  Copyright: 
//    (C) 2024 Thorsten Brach. All rights reserved                                                                         
//                                                                           
//  Disclaimer:                                                                           
//    This project is provided without any guarantee and can be used for   
//    private and commercial purposes. Any commercial use is at the user’s 
//    own risk and responsibility.
//
// -------------------------------------------------------------------------
TYPE TelegramPlcToRobFragmentHeader :
STRUCT
  /// Command Instance Identifier used to assign the CMD payload to a specific CMD instance
  ID             : UINT;
  /// Empty reserve byte
  Reserve        : BYTE;
  /// Fragment Action Byte
  FragmentAction : FragmentAction;
  /// Append received payload in the receive buffer at this position
  PayloadPointer : UINT;
  /// Length of the CMD payload
  PayloadLength  : UINT;  
END_STRUCT
END_TYPE

{attribute 'pack_mode' := '1'} 
// ------------------------------------------------------------------------- 
//  SRCI Robot Library                                                
// ------------------------------------------------------------------------- 
//                                                                           
//  Object:      TelegramPlcToRobHeader                                       
//  Author:      Thorsten Brach                                                
//  Date:        2024-06-01
//
//  Description:                                              
//   
//                                                                           
//  Copyright: 
//    (C) 2024 Thorsten Brach. All rights reserved                                                                         
//                                                                           
//  Disclaimer:                                                                           
//    This project is provided without any guarantee and can be used for   
//    private and commercial purposes. Any commercial use is at the user’s 
//    own risk and responsibility.
//
// -------------------------------------------------------------------------
TYPE TelegramPlcToRobHeader :
STRUCT
  /// Version of SRCI specification
  /// Bit 0-4 : Minor version = Features        (0..31)
  /// Bit 5-7 : Major version = Breaking change (0..07)
  SRCIVersion            : VersionStruct;
  /// Fast stop trigger 
  FastStop               : BYTE;
  /// Connection alive signal
  LifeSign               : BYTE;
  /// Number of Bytes of the frame to be used for the telegram of the given Axisgroup. Direction client to server
  TelegramLengthPlcToRob : UINT;
  /// Number of Bytes of the frame to be used for the telegram of the given Axisgroup. Direction server to client
  TelegramLengthRobToPlc : UINT;
  /// Control AxesGroupID Telegtam state control
  AxesGroupID            : BYTE;
  /// Telegtam state control
  Control                : ControlHalfByte;
  /// Reserved for later versions
  Reserved               : BYTE;
  /// Configuration of the optional cyclic data. Direction client to server
  TelegramNumberPlcToRob : UINT;
  /// Configuration of the optional cyclic data. Direction server to client
  TelegramNumberRobToPlc : UINT;
  /// Date of the client in the format days since 1990.01.01
  ClientDate             : IEC_DATE;
  /// Time in the clients time zone in the format milliseconds since start of day
  ClientTime             : IEC_TIME;  
END_STRUCT
END_TYPE

{attribute 'pack_mode' := '1'} 
// ------------------------------------------------------------------------- 
//  SRCI Robot Library                                                
// ------------------------------------------------------------------------- 
//                                                                           
//  Object:      TelegramPlcToRobSequence                                       
//  Author:      Thorsten Brach                                                
//  Date:        2024-06-01
//
//  Description:                                              
//   
//                                                                           
//  Copyright: 
//    (C) 2024 Thorsten Brach. All rights reserved                                                                         
//                                                                           
//  Disclaimer:                                                                           
//    This project is provided without any guarantee and can be used for   
//    private and commercial purposes. Any commercial use is at the user’s 
//    own risk and responsibility.
//
// -------------------------------------------------------------------------
TYPE TelegramPlcToRobSequence :
STRUCT
  /// Header
  Header   : TelegramPlcTorobSequenceHeader;
  /// Fragment
  Fragment : ARRAY[0..9] OF TelegramPlcToRobFragment;
END_STRUCT
END_TYPE

{attribute 'pack_mode' := '1'} 
// ------------------------------------------------------------------------- 
//  SRCI Robot Library                                                
// ------------------------------------------------------------------------- 
//                                                                           
//  Object:      TelegramPlcTorobSequenceHeader                                       
//  Author:      Thorsten Brach                                                
//  Date:        2024-06-01
//
//  Description:                                              
//   
//                                                                           
//  Copyright: 
//    (C) 2024 Thorsten Brach. All rights reserved                                                                         
//                                                                           
//  Disclaimer:                                                                           
//    This project is provided without any guarantee and can be used for   
//    private and commercial purposes. Any commercial use is at the user’s 
//    own risk and responsibility.
//
// -------------------------------------------------------------------------
TYPE TelegramPlcTorobSequenceHeader :
STRUCT
  /// Telegram Sequence and Acknowledgement number
  SEQ_ACK      : UINT;
  /// Length of the Telegram Sequence excluding this Telegram Sequence Header
  PayloadLength : UINT;
END_STRUCT
END_TYPE

{attribute 'pack_mode' := '1'} 
// ------------------------------------------------------------------------- 
//  SRCI Robot Library                                                
// ------------------------------------------------------------------------- 
//                                                                           
//  Object:      TelegramRobToPlcCyclicOptionalData                                       
//  Author:      Thorsten Brach                                                
//  Date:        2024-06-01
//
//  Description:                                              
//   
//                                                                           
//  Copyright: 
//    (C) 2024 Thorsten Brach. All rights reserved                                                                         
//                                                                           
//  Disclaimer:                                                                           
//    This project is provided without any guarantee and can be used for   
//    private and commercial purposes. Any commercial use is at the user’s 
//    own risk and responsibility.
//
// -------------------------------------------------------------------------
TYPE TelegramRobToPlcCyclicOptionalData :
STRUCT
    /// Transmit cyclic data from PLC to RC for the usage in a subprogram on the RC called via the function “CallSubprogram”
  SubProgramData        :  TelegramRobToPlcCyclicOptionalSubProgramData;
  /// cartesian position with TCP position (X, Y,Z), rotation (RX, RY, RZ), configuration bytes (Config, TurnNumber), position of first external axis (E1) and corresponding coordinate systems (ToolNo, FrameNo)
  CartesianPosition     :  TelegramRobToPlcCyclicOptionalCartesianPosition;
  /// axes position with joint values (J1, J2, J3,J4, J5, J6) and position of first external axis (E1)
  JointPosition         :  TelegramRobToPlcCyclicOptionalJointPosition;
  /// force with the divided forces in the individual directions (X, Y, Z, RX, RY, RZ)
  Force                 :  TelegramRobToPlcCyclicOptionalForce;
  /// Transmit actual axes current of individual axes (J1, J2, J3, J4, J5, J6)
  Current               :  TelegramRobToPlcCyclicOptionalCurrent;
  /// Set to 1 to define two Sequences in one Telegram. If activated, 
  /// 2 sequences also has to be activated in the ClientServer direction.
  TwoSequences          : BYTE;  
  /// Transmit the external axis values for an extended cartesian position (E2, E3, E4, E5, E6)
  /// When selected, Tool and Frame will automatically cyclically be sent from client to server.
  CartesianPositionExt  :  TelegramRobToPlcCyclicOptionalCartesianPositionExt;
  /// Transmit the external axis values for an extended joint position (E2, E3, E4, E5, E6)
  JointPositionExt      :  TelegramRobToPlcCyclicOptionalJointPositionExt;
  /// Transmit actual axes force of individual axes (E1, E2, E3, E4, E5, E6)
  ForceExt              :  TelegramRobToPlcCyclicOptionalCurrentExt;
  /// Transmit actual axes current of individual axes (E1, E2, E3, E4, E5, E6)
  CurrentExt            :  TelegramRobToPlcCyclicOptionalCurrentExt;
END_STRUCT
END_TYPE

{attribute 'pack_mode' := '1'} 
// ------------------------------------------------------------------------- 
//  SRCI Robot Library                                                
// ------------------------------------------------------------------------- 
//                                                                           
//  Object:      TelegramFooter                                       
//  Author:      Thorsten Brach                                                
//  Date:        2024-06-01
//
//  Description:                                              
//   
//                                                                           
//  Copyright: 
//    (C) 2024 Thorsten Brach. All rights reserved                                                                         
//                                                                           
//  Disclaimer:                                                                           
//    This project is provided without any guarantee and can be used for   
//    private and commercial purposes. Any commercial use is at the user’s 
//    own risk and responsibility.
//
// -------------------------------------------------------------------------
TYPE TelegramFooter :
STRUCT
  /// Bit 00: Connection alive signal
  LifeSign : BOOL;
  /// Bit 01 
  Bit01    : BOOL;
  /// Bit 02 
  Bit02    : BOOL;
  /// Bit 03 
  Bit03    : BOOL;
  /// Bit 04 
  Bit04    : BOOL;
  /// Bit 05 
  Bit05    : BOOL;
  /// Bit 06 
  Bit06    : BOOL;
  /// Bit 07 
  Bit07    : BOOL;    
END_STRUCT
END_TYPE

{attribute 'pack_mode' := '1'} 
// ------------------------------------------------------------------------- 
//  SRCI Robot Library                                                
// ------------------------------------------------------------------------- 
//                                                                           
//  Object:      TelegramRobToPlcCyclic                                       
//  Author:      Thorsten Brach                                                
//  Date:        2024-06-01
//
//  Description:                                              
//   
//                                                                           
//  Copyright: 
//    (C) 2024 Thorsten Brach. All rights reserved                                                                         
//                                                                           
//  Disclaimer:                                                                           
//    This project is provided without any guarantee and can be used for   
//    private and commercial purposes. Any commercial use is at the user’s 
//    own risk and responsibility.
//
// -------------------------------------------------------------------------
TYPE TelegramRobToPlcHeader :
STRUCT
  /// Version of SRCI specification
  /// Bit 0-4 : Minor version = Features        (0..31)
  /// Bit 5-7 : Major version = Breaking change (0..07)
  SRCIVersion   : VersionStruct;
  /// Connection alive signal
  LifeSign      : BYTE;
  /// Reserved byte
  Reserved      : BYTE;
  /// Initialization and Telegram control state
  TelegramState : USINT;
  /// Combination of various RA related states.
  StatusRobotArm: RaStatusWord;
  /// Actual override in percentage encoding 
  Override      : UINT;
END_STRUCT
END_TYPE

{attribute 'pack_mode' := '1'} 
// ------------------------------------------------------------------------- 
//  SRCI Robot Library                                                
// ------------------------------------------------------------------------- 
//                                                                           
//  Object:      TelegramPlcToRobCyclicOptionalCartesianPos                                       
//  Author:      Thorsten Brach                                                
//  Date:        2024-06-01
//
//  Description:                                              
//   
//                                                                           
//  Copyright: 
//    (C) 2024 Thorsten Brach. All rights reserved                                                                         
//                                                                           
//  Disclaimer:                                                                           
//    This project is provided without any guarantee and can be used for   
//    private and commercial purposes. Any commercial use is at the user’s 
//    own risk and responsibility.
//
// -------------------------------------------------------------------------
TYPE TelegramPlcToRobCyclicOptionalCartesianPosition :
STRUCT
  /// TCP Position on the X-Axis
  X          : REAL;
  /// TCP Position on the Y-Axis
  Y          : REAL;
  /// TCP Position on the Z-Axis
  Z          : REAL;
  /// Rotation around the X-Axis (RX)
  Rx         : REAL;
  /// Rotation around the Y-Axis (RY)
  Ry         : REAL;
  /// Rotation around the Z-Axis (RZ)
  Rz         : REAL;
  /// Configuration data of the robot (Config)
  Config     : ArmConfigParameter;
  /// Turn number of the axes (TurnNumber)
  TurnNumber : TurnNumber;
  /// Position of first external axis
  E1         : REAL;
END_STRUCT
END_TYPE

{attribute 'pack_mode' := '1'} 
// ------------------------------------------------------------------------- 
//  SRCI Robot Library                                                
// ------------------------------------------------------------------------- 
//                                                                           
//  Object:      TelegramPlcToRobCyclicOptionalCartesianPositionExt                                       
//  Author:      Thorsten Brach                                                
//  Date:        2024-06-01
//
//  Description:                                              
//   
//                                                                           
//  Copyright: 
//    (C) 2024 Thorsten Brach. All rights reserved                                                                         
//                                                                           
//  Disclaimer:                                                                           
//    This project is provided without any guarantee and can be used for   
//    private and commercial purposes. Any commercial use is at the user’s 
//    own risk and responsibility.
//
// -------------------------------------------------------------------------
TYPE TelegramPlcToRobCyclicOptionalCartesianPositionExt :
STRUCT
  /// Position of second external axis
  E2 : REAL;
  /// Position of third external axis
  E3 : REAL;
  /// Position of fourth external axis
  E4 : REAL;
  /// Position of fifth external axis
  E5 : REAL;
  /// Position of sixth external axis
  E6 : REAL;    
END_STRUCT
END_TYPE

{attribute 'pack_mode' := '1'} 
// ------------------------------------------------------------------------- 
//  SRCI Robot Library                                                
// ------------------------------------------------------------------------- 
//                                                                           
//  Object:      TelegramPlcToRobCyclicOptionalCurrent                                       
//  Author:      Thorsten Brach                                                
//  Date:        2024-06-01
//
//  Description:                                              
//   
//                                                                           
//  Copyright: 
//    (C) 2024 Thorsten Brach. All rights reserved                                                                         
//                                                                           
//  Disclaimer:                                                                           
//    This project is provided without any guarantee and can be used for   
//    private and commercial purposes. Any commercial use is at the user’s 
//    own risk and responsibility.
//
// -------------------------------------------------------------------------
TYPE TelegramPlcToRobCyclicOptionalCurrent :
STRUCT
  /// Current of first joint of the robot
  J1 : REAL;
  /// Current of second joint of the robot
  J2 : REAL;
  /// Current of third joint of the robot
  J3 : REAL;
  /// Current of fourth joint of the robot
  J4 : REAL;
  /// Current of fifth joint of the robot
  J5 : REAL;
  /// Current of sixth joint of the robot
  J6 : REAL;  
END_STRUCT
END_TYPE

{attribute 'pack_mode' := '1'} 
// ------------------------------------------------------------------------- 
//  SRCI Robot Library                                                
// ------------------------------------------------------------------------- 
//                                                                           
//  Object:      TelegramPlcToRobCyclicOptionalCurrentExt                                       
//  Author:      Thorsten Brach                                                
//  Date:        2024-06-01
//
//  Description:                                              
//   
//                                                                           
//  Copyright: 
//    (C) 2024 Thorsten Brach. All rights reserved                                                                         
//                                                                           
//  Disclaimer:                                                                           
//    This project is provided without any guarantee and can be used for   
//    private and commercial purposes. Any commercial use is at the user’s 
//    own risk and responsibility.
//
// -------------------------------------------------------------------------
TYPE TelegramPlcToRobCyclicOptionalCurrentExt :
STRUCT
  /// Current of first external joint of the robot
  E1 : REAL;
  /// Current of second external axis
  E2: REAL;
  /// Current of third external axis
  E3: REAL;
  /// Current of fourth external axis
  E4: REAL;
  /// Current of fifth external axis
  E5: REAL;
  /// Current of sixth external axis
  E6: REAL;  
END_STRUCT
END_TYPE

{attribute 'pack_mode' := '1'} 
// ------------------------------------------------------------------------- 
//  SRCI Robot Library                                                
// ------------------------------------------------------------------------- 
//                                                                           
//  Object:      TelegramPlcToRobCyclicOptionalForce                                       
//  Author:      Thorsten Brach                                                
//  Date:        2024-06-01
//
//  Description:                                              
//   
//                                                                           
//  Copyright: 
//    (C) 2024 Thorsten Brach. All rights reserved                                                                         
//                                                                           
//  Disclaimer:                                                                           
//    This project is provided without any guarantee and can be used for   
//    private and commercial purposes. Any commercial use is at the user’s 
//    own risk and responsibility.
//
// -------------------------------------------------------------------------
TYPE TelegramPlcToRobCyclicOptionalForce :
STRUCT
  /// Force on the X-Axis
  X : REAL;
  /// Force on the Y-Axis
  Y : REAL;
  /// Force on the Z-Axis
  Z : REAL;
  /// Force around the X-Axis (RX)
  Rx : REAL;
  /// Force around the Y-Axis (RY)
  Ry : REAL;
  /// Force around the Z-Axis (RZ)
  Rz : REAL;
END_STRUCT
END_TYPE

{attribute 'pack_mode' := '1'} 
// ------------------------------------------------------------------------- 
//  SRCI Robot Library                                                
// ------------------------------------------------------------------------- 
//                                                                           
//  Object:      TelegramPlcToRobCyclicOptionalForceExt                                       
//  Author:      Thorsten Brach                                                
//  Date:        2024-06-01
//
//  Description:                                              
//   
//                                                                           
//  Copyright: 
//    (C) 2024 Thorsten Brach. All rights reserved                                                                         
//                                                                           
//  Disclaimer:                                                                           
//    This project is provided without any guarantee and can be used for   
//    private and commercial purposes. Any commercial use is at the user’s 
//    own risk and responsibility.
//
// -------------------------------------------------------------------------
TYPE TelegramPlcToRobCyclicOptionalForceExt :
STRUCT
  /// Force on the external axis 1
  E1 : REAL;
  /// Force on the external axis 2
  E2 : REAL;
  /// Force on the external axis 3
  E3 : REAL;
  /// Force om the external axis 4
  E4 : REAL;
  /// Force on the external axis 5
  E5 : REAL;
  /// Force on the external axis 6
  E6 : REAL;
END_STRUCT
END_TYPE

{attribute 'pack_mode' := '1'} 
// ------------------------------------------------------------------------- 
//  SRCI Robot Library                                                
// ------------------------------------------------------------------------- 
//                                                                           
//  Object:      TelegramPlcToRobCyclicOptionalJointPosition                                       
//  Author:      Thorsten Brach                                                
//  Date:        2024-06-01
//
//  Description:                                              
//   
//                                                                           
//  Copyright: 
//    (C) 2024 Thorsten Brach. All rights reserved                                                                         
//                                                                           
//  Disclaimer:                                                                           
//    This project is provided without any guarantee and can be used for   
//    private and commercial purposes. Any commercial use is at the user’s 
//    own risk and responsibility.
//
// -------------------------------------------------------------------------
TYPE TelegramPlcToRobCyclicOptionalJointPosition :
STRUCT
  /// Position of first joint of the robot
  J1 : REAL;
  /// Position of second joint of the robot
  J2 : REAL;
  /// Position of third joint of the robot
  J3 : REAL;
  /// Position of fourth joint of the robot
  J4 : REAL;
  /// Position of fifth joint of the robot
  J5 : REAL;
  /// Position of sixth joint of the robot
  J6 : REAL;
  /// Position of first external axis 
  E1 : REAL;  
END_STRUCT
END_TYPE

{attribute 'pack_mode' := '1'} 
// ------------------------------------------------------------------------- 
//  SRCI Robot Library                                                
// ------------------------------------------------------------------------- 
//                                                                           
//  Object:      TelegramPlcToRobCyclicOptionalJointPositionExt                                       
//  Author:      Thorsten Brach                                                
//  Date:        2024-06-01
//
//  Description:                                              
//   
//                                                                           
//  Copyright: 
//    (C) 2024 Thorsten Brach. All rights reserved                                                                         
//                                                                           
//  Disclaimer:                                                                           
//    This project is provided without any guarantee and can be used for   
//    private and commercial purposes. Any commercial use is at the user’s 
//    own risk and responsibility.
//
// -------------------------------------------------------------------------
TYPE TelegramPlcToRobCyclicOptionalJointPositionExt :
STRUCT
  /// Position of second external axis
  E2: REAL;
  /// Position of third external axis
  E3: REAL;
  /// Position of fourth external axis
  E4: REAL;
  /// Position of fifth external axis
  E5: REAL;
  /// Position of sixth external axis
  E6: REAL;    
END_STRUCT
END_TYPE

{attribute 'pack_mode' := '1'} 
// ------------------------------------------------------------------------- 
//  SRCI Robot Library                                                
// ------------------------------------------------------------------------- 
//                                                                           
//  Object:      TelegramPlcToRobCyclicOptionalSubProgramData                                       
//  Author:      Thorsten Brach                                                
//  Date:        2024-06-01
//
//  Description:                                              
//   
//                                                                           
//  Copyright: 
//    (C) 2024 Thorsten Brach. All rights reserved                                                                         
//                                                                           
//  Disclaimer:                                                                           
//    This project is provided without any guarantee and can be used for   
//    private and commercial purposes. Any commercial use is at the user’s 
//    own risk and responsibility.
//
// -------------------------------------------------------------------------
TYPE TelegramPlcToRobCyclicOptionalSubProgramData :
STRUCT
  /// Sub program data
  Data : ARRAY [0..25] OF BYTE;
END_STRUCT
END_TYPE

{attribute 'pack_mode' := '1'} 
// ------------------------------------------------------------------------- 
//  SRCI Robot Library                                                
// ------------------------------------------------------------------------- 
//                                                                           
//  Object:      TelegramRobToPlcCyclicOptionalCartesianPosition                                       
//  Author:      Thorsten Brach                                                
//  Date:        2024-06-01
//
//  Description:                                              
//   
//                                                                           
//  Copyright: 
//    (C) 2024 Thorsten Brach. All rights reserved                                                                         
//                                                                           
//  Disclaimer:                                                                           
//    This project is provided without any guarantee and can be used for   
//    private and commercial purposes. Any commercial use is at the user’s 
//    own risk and responsibility.
//
// -------------------------------------------------------------------------
TYPE TelegramRobToPlcCyclicOptionalCartesianPosition :
STRUCT
  /// TCP Position on the X-Axis
  X                    : REAL;
  /// TCP Position on the Y-Axis
  Y                    : REAL;
  /// TCP Position on the Z-Axis
  Z                    : REAL;
  /// Rotation around the X-Axis (RX)
  Rx                   : REAL;
  /// Rotation around the Y-Axis (RY)
  Ry                   : REAL;
  /// Rotation around the Z-Axis (RZ)
  Rz                   : REAL;
  /// Configuration data of the robot (Config)
  Config               : ArmConfigParameter;
  /// Turn number of the axes (TurnNumber)
  TurnNumber           : TurnNumber;
  /// Position of first external axis
  E1                   : REAL;  
  /// Position of second external axis
  E2                   : REAL;
  /// Position of third external axis
  E3                   : REAL;
  /// Position of fourth external axis
  E4                   : REAL;
  /// Position of fifth external axis
  E5                   : REAL;
  /// Position of sixth external axis
  E6                   : REAL;      
  /// Tool Number
  ToolNo               : USINT;
  /// Frane Number
  FrameNo              : USINT;
  /// Currently used tool number
  CurrentlyUsedToolNo  : USINT;
  /// Currently used frame number
  CurrentlyUsedFrameNo : USINT;
  /// Reserve
  Reserve_1            : BYTE;
  /// Reserve
  Reserve_2            : BYTE;  
END_STRUCT
END_TYPE

